TYPE ST_EL3443_DPM_MUX_REAL :
STRUCT
    nSelector : UINT := E_EL3443_DPM_Phase.Error_INDEX_Not_Valid;
    fValueRef : REFERENCE TO REAL;
END_STRUCT
END_TYPE

(* stored: Version 1.1.0.1, ProductVersion 3.1.4024.12
   DUT ST_EL3443_DPM_MUX_REAL: Id {ee453e1c-8fff-4758-a1f8-ff37c138b1fb} *)
